{attribute 'qualified_only'}
{attribute 'strict'}
TYPE E_Horn :
(
	off := 0,
	beep,
	short,
	long
);
END_TYPE

(* stored: Version 1.1.0.1, ProductVersion 3.1.4024.15
   DUT E_Horn: Id {b033c196-a04e-49b0-90e9-2a923f9dd67c} *)
